// TwinCAT 3 PLC project Untitled1
// ProgramVersion: 3.1.4023.0
// libraries:
//   Tc2_Standard, * (Beckhoff Automation GmbH)
//   Tc2_System, * (Beckhoff Automation GmbH)
//   Tc3_Module, * (Beckhoff Automation GmbH)
// project tree:
//   / Class Diagram.TcCD (not stored), PlcTask.TcTTO
//   FBs/ Motor.TcPOU, DieselMotor.TcPOU, ElectricMotor.TcPOU, ElectricAdapterMotor.TcPOU, GasolineMotor.TcPOU
//   POUs/ MAIN.TcPOU
// real-time tasks:
//   TASK PlcTask: cycle T#10ms, priority 20, ADS port 350

CONFIGURATION Untitled1
    RESOURCE PLC ON TwinCAT3
        TASK PlcTask(INTERVAL := T#10ms, PRIORITY := 20);
        PROGRAM MAIN WITH PlcTask : MAIN;
    END_RESOURCE
END_CONFIGURATION

// ---- POUs/MAIN.TcPOU
PROGRAM MAIN
VAR
	gasolineMotor 				: GasolineMotor;
	dieselMotor 				: DieselMotor;
	electricAdapterMotor 		: ElectricAdapterMotor;
	
	bGasolineMotor 				: BOOL;
	bDieselMotor 				: BOOL;
	bElectricAdapterMotor 		: BOOL;
	
	
END_VAR

//Gasoline motor
IF bGasolineMotor THEN
	bGasolineMotor := FALSE;
	gasolineMotor.Startup();
	gasolineMotor.Speedup();
	gasolineMotor.Stop();
	gasolineMotor.LoadFuel();
END_IF


//Diesel motor
IF bDieselMotor THEN
	bDieselMotor := FALSE;
	dieselMotor.Startup();
	dieselMotor.Speedup();
	dieselMotor.Stop();
	dieselMotor.LoadFuel();
END_IF


//Electric motor
IF bElectricAdapterMotor THEN
	bElectricAdapterMotor := FALSE;
	electricAdapterMotor.Startup();
	electricAdapterMotor.Speedup();
	electricAdapterMotor.Stop();
	electricAdapterMotor.LoadFuel();
END_IF

END_PROGRAM

// ---- FBs/GasolineMotor.TcPOU
FUNCTION_BLOCK GasolineMotor EXTENDS Motor

METHOD PUBLIC LoadFuel
ADSLOGSTR(    msgCtrlMask:=ADSLOG_MSGTYPE_LOG,
              msgFmtStr:='Loading fuel into the Gasoline motor..',
              strArg:='');
END_METHOD

METHOD PUBLIC SpeedUp
ADSLOGSTR(    msgCtrlMask:=ADSLOG_MSGTYPE_LOG,
              msgFmtStr:='Accelerating the Gasoline motor...',
              strArg:='');
END_METHOD

METHOD PUBLIC StartUp
ADSLOGSTR(    msgCtrlMask:=ADSLOG_MSGTYPE_LOG,
              msgFmtStr:='Starting the Gasoline motor...',
              strArg:='');
END_METHOD

METHOD PUBLIC Stop
ADSLOGSTR(    msgCtrlMask:=ADSLOG_MSGTYPE_LOG,
              msgFmtStr:='Stopping the Gasoline motor...',
              strArg:='');
END_METHOD

END_FUNCTION_BLOCK

// ---- FBs/Motor.TcPOU
FUNCTION_BLOCK ABSTRACT Motor

METHOD PUBLIC ABSTRACT LoadFuel
END_METHOD

METHOD PUBLIC ABSTRACT SpeedUp
END_METHOD

METHOD PUBLIC ABSTRACT StartUp
END_METHOD

METHOD PUBLIC ABSTRACT Stop
END_METHOD

END_FUNCTION_BLOCK

// ---- FBs/DieselMotor.TcPOU
FUNCTION_BLOCK DieselMotor EXTENDS Motor

METHOD PUBLIC LoadFuel
ADSLOGSTR(    msgCtrlMask:=ADSLOG_MSGTYPE_LOG,
              msgFmtStr:='Loading fuel into the Diesel motor...',
              strArg:='');
END_METHOD

METHOD PUBLIC SpeedUp
ADSLOGSTR(    msgCtrlMask:=ADSLOG_MSGTYPE_LOG,
              msgFmtStr:='Accelerating the Diesel motor...',
              strArg:='');
END_METHOD

METHOD PUBLIC StartUp
ADSLOGSTR(    msgCtrlMask:=ADSLOG_MSGTYPE_LOG,
              msgFmtStr:='Starting the Diesel motor...',
              strArg:='');
END_METHOD

METHOD PUBLIC Stop
ADSLOGSTR(    msgCtrlMask:=ADSLOG_MSGTYPE_LOG,
              msgFmtStr:='Stopping the Diesel motor...',
              strArg:='');
END_METHOD

END_FUNCTION_BLOCK

// ---- FBs/ElectricAdapterMotor.TcPOU
{attribute 'enable_dynamic_creation'}
FUNCTION_BLOCK ElectricAdapterMotor EXTENDS Motor
VAR
	pElectricEngine : POINTER TO ElectricMotor;
END_VAR

METHOD FB_exit : BOOL
VAR_INPUT
	bInCopyCode : BOOL; // if TRUE, the exit method is called for exiting an instance that is copied afterwards (online change).
END_VAR
__DELETE (pElectricEngine);
END_METHOD


METHOD FB_init : BOOL
VAR_INPUT
	bInitRetains : BOOL; // if TRUE, the retain variables are initialized (warm start / cold start)
	bInCopyCode : BOOL;  // if TRUE, the instance afterwards gets moved into the copy code (online change)
END_VAR
pElectricEngine := __NEW(ElectricMotor);
END_METHOD

METHOD PUBLIC LoadFuel
pElectricEngine^.Plug();
END_METHOD

METHOD PUBLIC SpeedUp
pElectricEngine^.Travel();
END_METHOD

METHOD PUBLIC StartUp
pElectricEngine^.Connect();
pElectricEngine^.Activate();
END_METHOD

METHOD PUBLIC Stop
pElectricEngine^.Deactivate();
pElectricEngine^.Stop();
END_METHOD

END_FUNCTION_BLOCK

// ---- FBs/ElectricMotor.TcPOU
{attribute 'enable_dynamic_creation'}
FUNCTION_BLOCK ElectricMotor
VAR
	_bConnected : BOOL;
	_bActivated : BOOL;
	_bTraveling	: BOOL;
	
	
END_VAR

METHOD Activate
IF NOT _bConnected THEN
	
	ADSLOGSTR(	msgCtrlMask:=ADSLOG_MSGTYPE_LOG,
              	msgFmtStr:='Impossible to activate an electric motor already not connected!',
              	strArg:='');
			  
ELSE
	
	_bActivated := TRUE;
	
	ADSLOGSTR(	msgCtrlMask:=ADSLOG_MSGTYPE_LOG,
              	msgFmtStr:='electric motor activated!',
              	strArg:='');
END_IF
END_METHOD

METHOD Connect
IF _bConnected THEN
	
	ADSLOGSTR(	msgCtrlMask:=ADSLOG_MSGTYPE_LOG,
              	msgFmtStr:='Impossible to connect an electric motor already connected!',
              	strArg:='');
			  
ELSE
	
	ADSLOGSTR(	msgCtrlMask:=ADSLOG_MSGTYPE_LOG,
              	msgFmtStr:='electric motor connected!',
              	strArg:='');
				
	_bConnected := TRUE;
END_IF
END_METHOD

METHOD Deactivate
IF _bActivated THEN
	
	_bActivated := FALSE;
	
	ADSLOGSTR(	msgCtrlMask:=ADSLOG_MSGTYPE_LOG,
              	msgFmtStr:='Electric motor deactivated!',
              	strArg:='');
ELSE
	
	ADSLOGSTR(	msgCtrlMask:=ADSLOG_MSGTYPE_LOG,
              	msgFmtStr:='Impossible to deactivated an electric motor already connected!',
              	strArg:='');
				
END_IF
END_METHOD

METHOD Disconnect
IF _bConnected THEN
	
	_bConnected := FALSE;
		
	ADSLOGSTR(	msgCtrlMask:=ADSLOG_MSGTYPE_LOG,
              	msgFmtStr:='electric motor disconnected...',
              	strArg:='');
ELSE
		
	ADSLOGSTR(	msgCtrlMask:=ADSLOG_MSGTYPE_LOG,
              	msgFmtStr:='Impossible to disconnect an electric motor that is connected!',
              	strArg:='');
END_IF
END_METHOD

METHOD Plug
IF NOT _bActivated THEN
	
	_bActivated := FALSE;
	
	ADSLOGSTR(	msgCtrlMask:=ADSLOG_MSGTYPE_LOG,
              	msgFmtStr:='Electric motor plugging bateries...',
              	strArg:='');
ELSE
	

	
	ADSLOGSTR(	msgCtrlMask:=ADSLOG_MSGTYPE_LOG,
              	msgFmtStr:='Impossible to plug an electric motor!',
              	strArg:='');
END_IF
END_METHOD

METHOD Stop
IF _bTraveling THEN
	
	_bTraveling := FALSE;

	ADSLOGSTR(	msgCtrlMask:=ADSLOG_MSGTYPE_LOG,
              	msgFmtStr:='Stopping vehicle with electric motor...',
              	strArg:='');
ELSE
	
	_bActivated := TRUE;
	
	ADSLOGSTR(	msgCtrlMask:=ADSLOG_MSGTYPE_LOG,
              	msgFmtStr:='Impossible to stop an electric motor that is not traveling!',
              	strArg:='');
END_IF
END_METHOD

METHOD Travel
IF (_bConnected AND _bActivated) THEN
	
	_bTraveling := TRUE;
	
	ADSLOGSTR(	msgCtrlMask:=ADSLOG_MSGTYPE_LOG,
              	msgFmtStr:='Traveling vehicle with electric motor...',
              	strArg:='');
ELSE
	
	ADSLOGSTR(	msgCtrlMask:=ADSLOG_MSGTYPE_LOG,
              	msgFmtStr:='The electric motor must be connected and activated!',
              	strArg:='');
END_IF
END_METHOD

END_FUNCTION_BLOCK
